Fanuc TP program (LS listing): UP026.LS

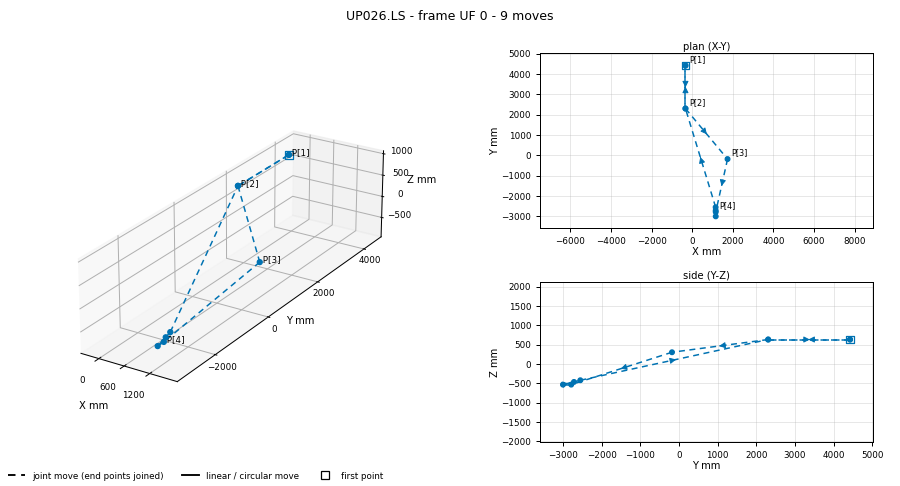
[picture p0: tool path of UP026.LS in frame UF 0, 9 of 9 moves have a stored position in this frame; points joined in program order, loops and branches not executed]
/PROG  UP026
/ATTR
OWNER		= MNEDITOR;
COMMENT		= "Ext. 1680 Pos. 2";
PROG_SIZE	= 4440;
CREATE		= DATE 23-07-11  TIME 01:05:54;
MODIFIED	= DATE 24-03-17  TIME 19:57:46;
FILE_NAME	= UP006;
VERSION		= 0;
LINE_COUNT	= 21;
MEMORY_SIZE	= 7936;
PROTECT		= READ_WRITE;
TCD:  STACK_SIZE	= 500,
      TASK_PRIORITY	= 50,
      TIME_SLICE	= 0,
      BUSY_LAMP_OFF	= 0,
      ABORT_REQUEST	= 0,
      PAUSE_REQUEST	= 0;
DEFAULT_GROUP	= 1,1,1,1,*;
CONTROL_CODE	= 00000000 00000000;
/APPL
/MN
   1:  UFRAME_NUM=0 ;
   2:  UTOOL_NUM=1 ;
   3:  PAYLOAD[2] ;
   4:  !Apagar Perfil Lib. 77 vs ST1680 ;
   5:J P[1] 100% CNT0 ACC100 TB    .10sec,P-SPS    ;
      1:  TC_ONLINE (ON) ;
      2:  DO[23]=OFF ;
      3:  TIMER[6]=RESET ;
      4:  TIMER[6]=START ;
      5:  CALL MAKRO050    ;
      6:  !Lib. de Herramientas ;
      7:  DO[43]=ON ;
      8:  DO[44]=ON ;
      9:  !Lib. de Anticolisiones ;
     10:  DO[80]=ON ;
     11:  DO[78]=OFF ;
     12:  DO[77]=ON ;
     13:  DO[75]=OFF ;
     14:  DO[74]=ON ;
     15:  DO[72]=OFF ;
     16:  !Apagar Pos. Base ;
     17:  DO[15]=OFF ;
     18:  !Robot en Trayectoria ;
     19:  DO[16]=ON ;
     20:  WAIT (DI[61] AND !DI[62] AND DI[76] AND M[1])    ;
     21:  DO[77]=OFF ;
     22:  WAIT (DI[23])    ;
     23:  DO[23]=ON ;
     24:  TC_ONLINE (DI[61] AND !DI[62] AND DI[76] AND M[1] AND M[30] AND M[32] AND M[33]) ;
       ------ ;
   6:J P[2] 100% CNT100 ACC100 TB   0.00sec,P-SPS    ;
      1:  TC_ONLINE (DI[61] AND !DI[62] AND DI[76] AND M[1] AND M[30] AND M[32] AND M[33]) ;
       ------ ;
   7:J P[3] 100% CNT100 ACC100 TB   0.00sec,P-SPS    ;
      1:  TC_ONLINE (DI[61] AND !DI[62] AND DI[76] AND M[1] AND M[30] AND M[32] AND M[33]) ;
       ------ ;
   8:J P[4] 100% CNT0 ACC100 TB    .10sec,P-SPS    ;
      1:  TC_ONLINE (ON) ;
      2:  DO[23]=OFF ;
      3:  WAIT (DI[23])    ;
      4:  DO[23]=ON ;
      5:  TC_ONLINE (DI[76] AND M[1] AND M[30] AND M[32] AND M[33]) ;
       ------ ;
   9:  !En Posicion ST1680-2 ;
  10:  !Dejar Pieza en ST1680-2 ;
  11:  !Fin de Trabajo 3 ;
  12:L P[5] 200mm/sec CNT0 ACC100 TB    .10sec,P-SPS    ;
      1:  TC_ONLINE (ON) ;
      2:  DO[23]=OFF ;
      3:  DO[75]=ON ;
      4:  WAIT (!DI[61] AND DI[62])    ;
      5:  F[2]=(ON) ;
      6:  CALL MAKRO343    ;
      7:  WAIT (M[34])    ;
      8:  F[1]=(ON) ;
      9:  CALL MAKRO342    ;
     10:  CALL MAKRO340    ;
     11:  WAIT (M[31])    ;
     12:  CALL MAKRO003    ;
     13:  GO[21]=2 ;
     14:  WAIT (DI[76])    ;
     15:  DO[75]=OFF ;
     16:  WAIT (DI[23])    ;
     17:  DO[23]=ON ;
     18:  TC_ONLINE (!DI[61] AND DI[62] AND DI[76] AND M[30] AND M[31] AND M[34]) ;
       ------ ;
  13:  PAYLOAD[1] ;
  14:L P[6] 300mm/sec CNT0 ACC100 TB    .10sec,P-SPS    ;
      1:  TC_ONLINE (ON) ;
      2:  DO[23]=OFF ;
      3:  WAIT (M[2])    ;
      4:  WAIT (DI[23])    ;
      5:  DO[23]=ON ;
      6:  TC_ONLINE (!DI[61] AND DI[62] AND DI[76] AND M[2] AND M[30] AND M[31] AND M[34]) ;
       ------ ;
  15:   ;
  16:  OVERRIDE=100% ;
  17:   ;
  18:J P[7] 70% CNT80 ACC75 TB   0.00sec,P-SPS    ;
      1:  TC_ONLINE (!DI[61] AND DI[62] AND DI[76] AND M[2] AND M[30] AND M[31] AND M[34]) ;
       ------ ;
  19:J P[8] 70% CNT80 ACC50 TB   0.00sec,P-SPS    ;
      1:  TC_ONLINE (!DI[61] AND DI[62] AND DI[76] AND M[2] AND M[30] AND M[31] AND M[34]) ;
       ------ ;
  20:  !Encender Perfil Lib 77 vs ST1680 ;
  21:J P[9] 80% CNT0 ACC50 TB    .10sec,P-SPS    ;
      1:  TC_ONLINE (ON) ;
      2:  DO[23]=OFF ;
      3:  TIMER[6]=STOP ;
      4:  F[2]=(ON) ;
      5:  CALL MAKRO342    ;
      6:  CALL MAKRO340    ;
      7:  WAIT (M[33])    ;
      8:  WAIT (DI[23])    ;
      9:  DO[23]=ON ;
     10:  TC_ONLINE (M[2] AND M[30] AND M[31] AND M[33]) ;
       ------ ;
/POS
P[1]{
   GP1:
	UF : 0, UT : 1,		CONFIG : 'F U T, 0, 0, 0',
	X =  -332.978  mm,	Y =  4426.811  mm,	Z =   636.000  mm,
	W =    91.999 deg,	P =      .001 deg,	R =  -180.000 deg,
	E1=  2500.000  mm
   GP2:
	UF : 0, UT : 1,
	J1=     0.000  mm
   GP3:
	UF : 0, UT : 1,
	J1=     0.000  mm
   GP4:
	UF : 0, UT : 1,
	J1=     0.000  mm
};
P[2]{
   GP1:
	UF : 0, UT : 1,		CONFIG : 'F U T, 0, 0, 0',
	X =  -332.978  mm,	Y =  2308.572  mm,	Z =   636.000  mm,
	W =    91.999 deg,	P =     0.000 deg,	R =   180.000 deg,
	E1=   381.761  mm
   GP2:
	UF : 0, UT : 1,
	J1=     0.000  mm
   GP3:
	UF : 0, UT : 1,
	J1=     0.000  mm
   GP4:
	UF : 0, UT : 1,
	J1=     0.000  mm
};
P[3]{
   GP1:
	UF : 0, UT : 1,		CONFIG : 'F U T, 0, 0, 0',
	X =  1739.657  mm,	Y =  -180.418  mm,	Z =   306.742  mm,
	W =   -92.319 deg,	P =    30.439 deg,	R =   -86.555 deg,
	E1=   -15.208  mm
   GP2:
	UF : 0, UT : 1,
	J1=     0.000  mm
   GP3:
	UF : 0, UT : 1,
	J1=     0.000  mm
   GP4:
	UF : 0, UT : 1,
	J1=     0.000  mm
};
P[4]{
   GP1:
	UF : 0, UT : 1,		CONFIG : 'F U T, 0, 0, 0',
	X =  1158.199  mm,	Y = -2787.980  mm,	Z =  -530.947  mm,
	W =   -90.023 deg,	P =    14.451 deg,	R =   -89.752 deg,
	E1=   -67.649  mm
   GP2:
	UF : 0, UT : 1,
	J1=     0.000  mm
   GP3:
	UF : 0, UT : 1,
	J1=     0.000  mm
   GP4:
	UF : 0, UT : 1,
	J1=     0.000  mm
};
P[5]{
   GP1:
	UF : 0, UT : 1,		CONFIG : 'F U T, 0, 0, 0',
	X =  1158.199  mm,	Y = -3001.575  mm,	Z =  -530.947  mm,
	W =   -90.023 deg,	P =    14.451 deg,	R =   -89.752 deg,
	E1=   -67.649  mm
   GP2:
	UF : 0, UT : 1,
	J1=     0.000  mm
   GP3:
	UF : 0, UT : 1,
	J1=     0.000  mm
   GP4:
	UF : 0, UT : 1,
	J1=     0.000  mm
};
P[6]{
   GP1:
	UF : 0, UT : 1,		CONFIG : 'F U T, 0, 0, 0',
	X =  1155.786  mm,	Y = -2716.474  mm,	Z =  -461.517  mm,
	W =   -90.120 deg,	P =    14.539 deg,	R =   -89.705 deg,
	E1=   -67.744  mm
   GP2:
	UF : 0, UT : 1,
	J1=     0.000  mm
   GP3:
	UF : 0, UT : 1,
	J1=     0.000  mm
   GP4:
	UF : 0, UT : 1,
	J1=     0.000  mm
};
P[7]{
   GP1:
	UF : 0, UT : 1,		CONFIG : 'F U T, 0, 0, 0',
	X =  1153.641  mm,	Y = -2552.350  mm,	Z =  -418.125  mm,
	W =   -89.375 deg,	P =    14.499 deg,	R =   -88.429 deg,
	E1=   -69.654  mm
   GP2:
	UF : 0, UT : 1,
	J1=     0.000  mm
   GP3:
	UF : 0, UT : 1,
	J1=     0.000  mm
   GP4:
	UF : 0, UT : 1,
	J1=     0.000  mm
};
P[8]{
   GP1:
	UF : 0, UT : 1,		CONFIG : 'F U T, 0, 0, 0',
	X =  -332.978  mm,	Y =  2308.572  mm,	Z =   636.000  mm,
	W =    91.999 deg,	P =     0.000 deg,	R =  -180.000 deg,
	E1=   381.761  mm
   GP2:
	UF : 0, UT : 1,
	J1=     0.000  mm
   GP3:
	UF : 0, UT : 1,
	J1=     0.000  mm
   GP4:
	UF : 0, UT : 1,
	J1=     0.000  mm
};
P[9]{
   GP1:
	UF : 0, UT : 1,		CONFIG : 'F U T, 0, 0, 0',
	X =  -332.978  mm,	Y =  4426.811  mm,	Z =   636.000  mm,
	W =    91.999 deg,	P =      .001 deg,	R =  -180.000 deg,
	E1=  2500.000  mm
   GP2:
	UF : 0, UT : 1,
	J1=     0.000  mm
   GP3:
	UF : 0, UT : 1,
	J1=     0.000  mm
   GP4:
	UF : 0, UT : 1,
	J1=     0.000  mm
};
/END
